ABB RobotStudio station: 210021601076.rspag

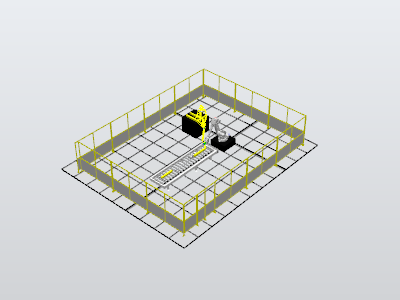
--- station ---
Station Aslam (saved by RobotStudio 23.2.10478.1)
Controller Controller2, task T_ROB1: task frame (RAPID world) sits at (580.05, 27.7, 395.4) mm, rotated rx 0 ry 0 rz 0.37 deg in the station
Controller Controller2
  mechanical unit ROB_1: IRB4600_40_255_C_01, 6 joints, base frame (0, 0, 0) mm
Layout (positions relative to the parent item):
  - Smart_Gripper_Servo_One_Vacuum [mechanism, from %ABB.RobotStudio.Models.SmartGripper%\ABB_Smart_Gripper_Servo_One_Vacuum.rslib] at (1934.43, -88.9, 888.73) mm, rotated rx -166.7 ry 89.28 rz -166.28 deg; joint values [0] (rad or m)
  - Conveyer [part, from %ABB.RobotStudio.Models.Conveyors%\Conveyor 950 4000 h2.rslib] at (1600, -500, 0) mm
  - Base [part] at (-3.62, 631.17, 0) mm, rotated rx 0 ry 0 rz 0.33 deg, size 1000 x 1000 x 400 mm
  - Box [part], size 800 x 100 x 100 mm
  - Conveyer [smart component]
      signals: DI movel, DO indic
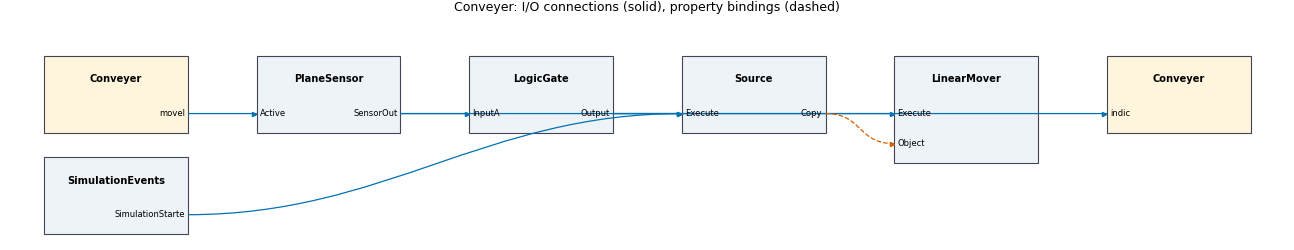
      connections:
        Conveyer.movel -> PlaneSensor.Active
        PlaneSensor.SensorOut -> Conveyer.indic
        PlaneSensor.SensorOut -> LogicGate.InputA
        LogicGate.Output -> LinearMover.Execute
        LogicGate.Output -> Source.Execute
        SimulationEvents.SimulationStarted -> Source.Execute
        Source.Copy => LinearMover.Object
    - PlaneSensor [smart component, from Components\PlaneSensor.rslib] at (1568.3, 52.45, 0) mm
        properties: Origin=[0.238634878927635 0.29755427370953 0.425]; Axis1=[0.1 0 0.1]; Axis2=[0 -0.77 0]; Tag=(none); SensedPart=Box_18
      - _sensorPart_ [part], size 100 x 770 x 100 mm
    - Source [smart component, from Components\Source.rslib]
        properties: Source=Box; Copy=Box_18; Parent=(none); Position=[0 0 0]; Orientation=[0 0 0]; Transient=false; PhysicsBehavior=-1
    - LinearMover [smart component, from Components\LinearMover.rslib]
        properties: Object=Box_18; Direction=[-3 0 0]; Speed=1; Reference=Global; ReferenceObject=(none)
    - LogicGate [smart component, from Components\LogicGate.rslib]
        properties: Operator=NOT; Delay=0
    - SimulationEvents [smart component, from Components\SimulationEvents.rslib]
  - AttachDetach [smart component]
      signals: DI attach, DO do
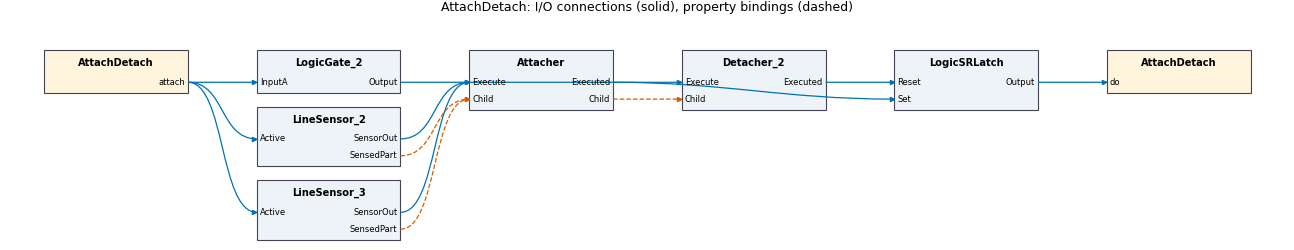
      connections:
        AttachDetach.attach -> LogicGate_2.InputA
        AttachDetach.attach -> LineSensor_2.Active
        LineSensor_2.SensorOut -> Attacher.Execute
        Detacher_2.Executed -> LogicSRLatch.Reset
        Attacher.Executed -> LogicSRLatch.Set
        LogicSRLatch.Output -> AttachDetach.do
        LogicGate_2.Output -> Detacher_2.Execute
        AttachDetach.attach -> LineSensor_3.Active
        LineSensor_3.SensorOut -> Attacher.Execute
        LineSensor_2.SensedPart => Attacher.Child
        Attacher.Child => Detacher_2.Child
        LineSensor_3.SensedPart => Attacher.Child
    - Attacher [smart component, from Components\Attacher.rslib]
        properties: Parent=Smart_Gripper_Servo_One_Vacuum; Flange=1; Child=Box_17; Mount=false; Offset=[0 0 0]; Orientation=[0 0 0]
    - Detacher_2 [smart component, from Components\Detacher.rslib]
        properties: Child=Box_17; KeepPosition=true
    - LogicSRLatch [smart component, from Components\LogicSRLatch.rslib]
    - LogicGate_2 [smart component, from Components\LogicGate.rslib]
        properties: Operator=NOT; Delay=0
    - LineSensor_3 [smart component, from Components\LineSensor.rslib] at (1971.18, -70.27, 838.23) mm, rotated rx -179.84 ry -0.7 rz -179.57 deg
        properties: Start=[0 0 0]; End=[0 0 0.02]; Length=0.02; Radius=0.0005; Tag=(none); SensedPart=Box_17; SensedPoint=[0.551275024414063 -1.6518037109375 1.09683813476563]
      - _sensorPart_ [part], size 1 x 1 x 20 mm
  - Box_ref2 [part] at (-4421.56, -1482.88, 580.2) mm, rotated rx 0 ry 0 rz -0.2 deg, size 800 x 100 x 100 mm
  - Place_box [part] at (0, -2580.03, 0) mm, size 1100 x 1100 x 1000 mm
  - Box_ref [part] at (986.59, 2917.03, 580.2) mm, rotated rx 0 ry 0 rz -90.6 deg, size 800 x 100 x 100 mm
  - IRB4600_40_255_C_01 [mechanism, from %ABB.RobotStudio.Models.IRB4600%\IRB4600_40_255_C_G_01.rslib] at (580.05, 27.7, 395.4) mm, rotated rx 0 ry 0 rz 0.37 deg; joint values [-0.1026, 0.2903, 0.8053, -3.2587, 1.0862, 3.1922] (rad or m)
  - Box_7 [part], size 800 x 100 x 100 mm
  - Box_9 [part], size 800 x 100 x 100 mm
  - Box_1 [part], size 800 x 100 x 100 mm
  - Box_3 [part], size 800 x 100 x 100 mm
  - Box_4 [part] at (638.69, 2911.14, 517.63) mm, rotated rx 0.12 ry -0.74 rz -90.21 deg, size 800 x 100 x 100 mm
  - Box_6 [part], size 800 x 100 x 100 mm
  - Box_7 [part], size 800 x 100 x 100 mm
  - Box_8 [part] at (-4416.13, -1490.91, 542.63) mm, rotated rx 0.37 ry -0.47 rz -0.11 deg, size 800 x 100 x 100 mm
  - Box_9 [part] at (953.48, 2910.35, 521.52) mm, rotated rx 0.12 ry -0.74 rz -90.21 deg, size 800 x 100 x 100 mm
  - Fence_2500 [graphiccomponentgroup, from Equipment\Fence_2500.rslib] at (-2465.89, 934.33, 0) mm
    - Body 1 [part, from Equipment\Fence_2500.rslib]
    - Body 2 [part, from Equipment\Fence_2500.rslib]
  - Fence_2500_2 [graphiccomponentgroup, from Equipment\Fence_2500.rslib] at (-2458.15, -1574.69, -2.82) mm
    - Body 1 [part, from Equipment\Fence_2500.rslib]
    - Body 2 [part, from Equipment\Fence_2500.rslib]
  - Fence_2500_3 [graphiccomponentgroup, from Equipment\Fence_2500.rslib] at (-2458.94, -4084.22, 0) mm
    - Body 1 [part, from Equipment\Fence_2500.rslib]
    - Body 2 [part, from Equipment\Fence_2500.rslib]
  - Fence_2500_4 [graphiccomponentgroup, from Equipment\Fence_2500.rslib] at (112.46, -4080.59, 0) mm, rotated rx 0 ry 0 rz -90 deg
    - Body 1 [part, from Equipment\Fence_2500.rslib]
    - Body 2 [part, from Equipment\Fence_2500.rslib]
  - Fence_2500_5 [graphiccomponentgroup, from Equipment\Fence_2500.rslib] at (2616.81, -4080.59, 0) mm, rotated rx 0 ry 0 rz -90 deg
    - Body 1 [part, from Equipment\Fence_2500.rslib]
    - Body 2 [part, from Equipment\Fence_2500.rslib]
  - Fence_2500_6 [graphiccomponentgroup, from Equipment\Fence_2500.rslib] at (-2390.88, -4080.59, 0) mm, rotated rx 0 ry 0 rz -90 deg
    - Body 1 [part, from Equipment\Fence_2500.rslib]
    - Body 2 [part, from Equipment\Fence_2500.rslib]
  - Fence_2500_7 [graphiccomponentgroup, from Equipment\Fence_2500.rslib] at (7575.33, -4087.76, 0) mm, rotated rx 0 ry 0 rz 90 deg
    - Body 1 [part, from Equipment\Fence_2500.rslib]
    - Body 2 [part, from Equipment\Fence_2500.rslib]
  - Fence_2500_8 [graphiccomponentgroup, from Equipment\Fence_2500.rslib] at (7396.23, 964.23, 0) mm
    - Body 1 [part, from Equipment\Fence_2500.rslib]
    - Body 2 [part, from Equipment\Fence_2500.rslib]
  - Fence_2500_9 [graphiccomponentgroup, from Equipment\Fence_2500.rslib] at (7396.23, -1514.89, 0) mm
    - Body 1 [part, from Equipment\Fence_2500.rslib]
    - Body 2 [part, from Equipment\Fence_2500.rslib]
  - Fence_2500_10 [graphiccomponentgroup, from Equipment\Fence_2500.rslib] at (7396.23, -4035.95, 0) mm
    - Body 1 [part, from Equipment\Fence_2500.rslib]
    - Body 2 [part, from Equipment\Fence_2500.rslib]
  - Gate [graphiccomponentgroup, from Equipment\Fence_Gate.rslib] at (5874.56, 3415.05, 0) mm, rotated rx 0 ry 0 rz -90 deg
    - Body 1 [part, from Equipment\Fence_Gate.rslib]
    - Body 2 [part, from Equipment\Fence_Gate.rslib]
    - Body 3 [part, from Equipment\Fence_Gate.rslib]
  - Fence_2500_11 [graphiccomponentgroup, from Equipment\Fence_2500.rslib] at (-2421.34, 3391.49, 0) mm, rotated rx 0 ry 0 rz -90 deg
    - Body 1 [part, from Equipment\Fence_2500.rslib]
    - Body 2 [part, from Equipment\Fence_2500.rslib]
  - Fence_2500_12 [graphiccomponentgroup, from Equipment\Fence_2500.rslib] at (112.89, 3391.49, 0) mm, rotated rx 0 ry 0 rz -90 deg
    - Body 1 [part, from Equipment\Fence_2500.rslib]
    - Body 2 [part, from Equipment\Fence_2500.rslib]
  - Fence_2500_13 [graphiccomponentgroup, from Equipment\Fence_2500.rslib] at (2639.04, 3391.49, 0) mm, rotated rx 0 ry 0 rz -90 deg
    - Body 1 [part, from Equipment\Fence_2500.rslib]
    - Body 2 [part, from Equipment\Fence_2500.rslib]
  - Fence_740_2 [graphiccomponentgroup, from Equipment\Fence_740.rslib] at (5139.35, 3403.98, 0) mm, rotated rx 0 ry 0 rz -90 deg
    - Body 1 [part, from Equipment\Fence_740.rslib]
    - Body 2 [part, from Equipment\Fence_740.rslib]
  - Box_13 [part], size 800 x 100 x 100 mm
  - Box_14 [part] at (-2520, 0, 0) mm, size 800 x 100 x 100 mm
  - Box_15 [part] at (-4416.13, -1490.91, 542.63) mm, rotated rx 0.37 ry -0.47 rz -0.11 deg, size 800 x 100 x 100 mm
  - Box_16 [part] at (953.48, 2910.35, 521.52) mm, rotated rx 0.12 ry -0.74 rz -90.21 deg, size 800 x 100 x 100 mm
  - Box_17 [part] at (638.69, 2911.14, 517.63) mm, rotated rx 0.12 ry -0.74 rz -90.21 deg, size 800 x 100 x 100 mm
  - Box_18 [part] at (-2664, 0, 0) mm, size 800 x 100 x 100 mm
Attachment: LineSensor_3 is attached to Smart_Gripper_Servo_One_Vacuum / DownFinger
Attachment: Smart_Gripper_Servo_One_Vacuum is attached to IRB4600_40_255_C_01 / Link6
Station logic (signal -> signal, property => property):
  Controller2.out -> AttachDetach.attach
  Controller2.di_output -> Conveyer.movel
  Conveyer.indic -> Controller2.start

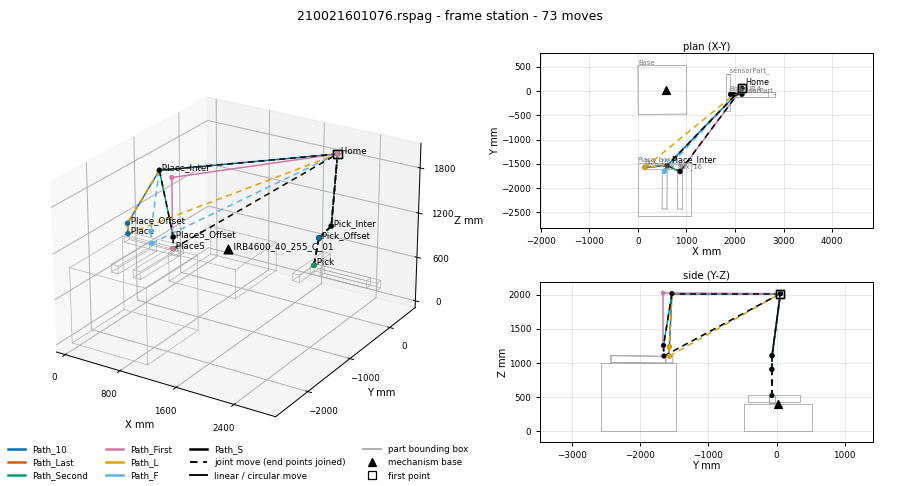
[picture p0: tool path of 210021601076.rspag in frame station, 73 of 73 moves have a stored position in this frame; points joined in program order, loops and branches not executed]
--- Controller Data/Controller2/RAPID/TASK1/PROGMOD/CalibData.mod ---
MODULE CalibData
    PERS tooldata Servo:=[TRUE,[[0,0,84],[1,0,0,0]],[0.226,[8.9,12.3,48.7],[1,0,0,0],0.00021,0.00024,0.00009]];
    PERS tooldata VaccumOne:=[TRUE,[[63.5,18.5,37.5],[0.707106781,0,0.707106781,0]],[0.226,[8.9,12.3,48.7],[1,0,0,0],0.00021,0.00024,0.00009]];
ENDMODULE

--- Controller Data/Controller2/RAPID/TASK1/PROGMOD/Module1.mod ---
MODULE Module1
        CONST robtarget Home:=[[1562.639382153,18.5,1623.75738686],[0.258819046,0,-0.965925826,0],[-1,-1,0,1],[9E+09,9E+09,9E+09,9E+09,9E+09,9E+09]];
    CONST robtarget Pick:=[[1325.709206308,-105.69931637,127.507161245],[0.005604326,-0.000424517,-0.99998295,0.001584379],[-1,-3,2,0],[9E+09,9E+09,9E+09,9E+09,9E+09,9E+09]];
    CONST robtarget Pick_Inter:=[[1561.851467861,-103.162107412,713.081838562],[0.258819024,0,-0.965925832,0],[-1,-3,2,0],[9E+09,9E+09,9E+09,9E+09,9E+09,9E+09]];
    CONST robtarget Pick_Offset:=[[1391.779201858,-106.126964158,512.226578953],[0.005604378,-0.000424533,-0.99998295,0.001584379],[-1,-3,2,0],[9E+09,9E+09,9E+09,9E+09,9E+09,9E+09]];
    CONST robtarget Place_Inter:=[[11.867363508,-1562.703465576,1623.756983637],[0.182623873,-0.68446068,-0.681561662,-0.183400653],[-2,-3,2,1],[9E+09,9E+09,9E+09,9E+09,9E+09,9E+09]];
    CONST robtarget Place:=[[-440.70574459,-1597.548111643,707.1200986],[0.001483954,-0.00137647,-0.999996574,-0.001659987],[-2,-2,0,1],[9E+09,9E+09,9E+09,9E+09,9E+09,9E+09]];
    CONST robtarget Place_Offset:=[[-444.124698969,-1597.525985837,843.908044243],[0.001483948,-0.001376451,-0.999996574,-0.001659976],[-2,-2,0,1],[9E+09,9E+09,9E+09,9E+09,9E+09,9E+09]];
    CONST robtarget PlaceS_Offset:=[[280.069318323,-1687.384959127,863.62826548],[0.000238405,0.708711216,0.705497899,-0.001034476],[-1,-2,1,0],[9E+09,9E+09,9E+09,9E+09,9E+09,9E+09]];
    CONST robtarget PlaceS:=[[275.144596365,-1682.104959802,708.235040947],[0.000238464,0.708711109,0.705498006,-0.001034365],[-1,-2,1,0],[9E+09,9E+09,9E+09,9E+09,9E+09,9E+09]];
    CONST robtarget PlaceF_Inter:=[[275.646442284,-1694.12601053,1633.167957717],[0.000238738,0.70871119,0.705497925,-0.00103415],[-1,-4,3,1],[9E+09,9E+09,9E+09,9E+09,9E+09,9E+09]];
    CONST robtarget PlaceF_Offset:=[[275.646447462,-1694.126005121,854.024783097],[0.000238763,0.708711188,0.705497927,-0.001034117],[-1,-4,3,1],[9E+09,9E+09,9E+09,9E+09,9E+09,9E+09]];
    CONST robtarget Place_F:=[[275.686493171,-1687.929599777,709.019601147],[0.000238779,0.708711216,0.705497899,-0.001034127],[-1,-4,3,1],[9E+09,9E+09,9E+09,9E+09,9E+09,9E+09]];
    CONST robtarget Place2_Offset:=[[-43.343867547,-1685.291053434,863.62834295],[0.000238739,0.708711198,0.705497917,-0.001034153],[-2,-3,2,0],[9E+09,9E+09,9E+09,9E+09,9E+09,9E+09]];
    CONST robtarget Place2:=[[-39.637509275,-1679.274249515,704.345546214],[0.000238825,0.708711224,0.705497891,-0.001034082],[-2,-3,2,0],[9E+09,9E+09,9E+09,9E+09,9E+09,9E+09]];
!***********************************************************
    !
    ! Module:  Module1
    !
    ! Description:
    !   <Insert description here>
    !
    ! Author: shahu
    !
    ! Version: 1.0
    !
    !***********************************************************


    !***********************************************************
    !
    ! Procedure main
    !
    !   This is the entry point of your program
    !
    !***********************************************************
    PROC main()
        !Add your code here
    ENDPROC
    PROC Path_10()
        MoveJ Home,v1000,z100,VaccumOne\WObj:=wobj0;
        MoveJ Pick_Inter,v1000,z100,VaccumOne\WObj:=wobj0;
        MoveJ Pick_Offset,v1000,z100,VaccumOne\WObj:=wobj0;
        MoveJ Pick,v1000,z100,VaccumOne\WObj:=wobj0;
        MoveJ Pick_Offset,v1000,z100,VaccumOne\WObj:=wobj0;
        MoveJ Pick_Inter,v1000,z100,VaccumOne\WObj:=wobj0;
        MoveJ Home,v1000,z100,VaccumOne\WObj:=wobj0;
        MoveL Place_Inter,v1000,z100,VaccumOne\WObj:=wobj0;
        MoveL Place_Offset,v1000,z100,VaccumOne\WObj:=wobj0;
        MoveL Place,v1000,z100,VaccumOne\WObj:=wobj0;
    ENDPROC
    PROC Path_Last()
        MoveJ Home,v1000,z100,VaccumOne\WObj:=wobj0;
        MoveJ Pick_Inter,v1000,z100,VaccumOne\WObj:=wobj0;
        MoveJ Pick_Offset,v1000,z100,VaccumOne\WObj:=wobj0;
        MoveJ Pick,v1000,z100,VaccumOne\WObj:=wobj0;
        MoveJ Pick_Offset,v1000,z100,VaccumOne\WObj:=wobj0;
        MoveJ Pick_Inter,v1000,z100,VaccumOne\WObj:=wobj0;
        MoveJ Home,v1000,z100,VaccumOne\WObj:=wobj0;
        MoveJ Place_Inter,v1000,z100,VaccumOne\WObj:=wobj0;
        MoveJ Place_Offset,v1000,z100,VaccumOne\WObj:=wobj0;
        MoveJ Place,v1000,z100,VaccumOne\WObj:=wobj0;
    ENDPROC
    PROC Path_Second()
        MoveJ Home,v1000,z100,VaccumOne\WObj:=wobj0;
        MoveJ Pick_Inter,v1000,z100,VaccumOne\WObj:=wobj0;
        MoveJ Pick_Offset,v1000,z100,VaccumOne\WObj:=wobj0;
        MoveJ Pick,v1000,z100,VaccumOne\WObj:=wobj0;
        MoveJ Pick_Offset,v1000,z100,VaccumOne\WObj:=wobj0;
        MoveJ Pick_Inter,v1000,z100,VaccumOne\WObj:=wobj0;
        MoveJ Home,v1000,z100,VaccumOne\WObj:=wobj0;
        MoveJ Place_Inter,v1000,z100,VaccumOne\WObj:=wobj0;
        MoveL PlaceS_Offset,v1000,z100,VaccumOne\WObj:=wobj0;
        MoveJ PlaceS,v1000,z100,VaccumOne\WObj:=wobj0;
    ENDPROC
    PROC Path_First()
        MoveJ Home,v1000,z100,VaccumOne\WObj:=wobj0;
        MoveJ Pick_Inter,v1000,z100,VaccumOne\WObj:=wobj0;
        MoveJ Pick_Offset,v1000,z100,VaccumOne\WObj:=wobj0;
        MoveJ Pick,v1000,z100,VaccumOne\WObj:=wobj0;
        MoveJ Pick_Offset,v1000,z100,VaccumOne\WObj:=wobj0;
        MoveJ Pick_Inter,v1000,z100,VaccumOne\WObj:=wobj0;
        MoveJ Home,v1000,z100,VaccumOne\WObj:=wobj0;
        MoveL PlaceF_Inter,v1000,z100,VaccumOne\WObj:=wobj0;
        MoveL PlaceF_Offset,v1000,z100,VaccumOne\WObj:=wobj0;
        MoveJ Place_F,v1000,z100,VaccumOne\WObj:=wobj0;
    ENDPROC
    PROC Final_Path()
        Path_F;
        Path_L;
        Path_S;

    ENDPROC
    PROC Path_L()
        MoveJ Home,v1000,z100,VaccumOne\WObj:=wobj0;
        MoveJ Pick_Inter,v1000,z100,VaccumOne\WObj:=wobj0;
        MoveJ Pick_Offset,v1000,z100,VaccumOne\WObj:=wobj0;
        MoveJ Pick,v1000,z100,VaccumOne\WObj:=wobj0;
        WaitTime 1;
        SetDO out,1;
        WaitTime 1;
        MoveJ Pick_Offset,v1000,z100,VaccumOne\WObj:=wobj0;
        MoveJ Pick_Inter,v1000,z100,VaccumOne\WObj:=wobj0;
        MoveJ Home,v1000,z100,VaccumOne\WObj:=wobj0;
        MoveJ Place_Inter,v1000,z100,VaccumOne\WObj:=wobj0;
        MoveJ Place_Offset,v1000,z100,VaccumOne\WObj:=wobj0;
        MoveJ Place,v1000,z100,VaccumOne\WObj:=wobj0;
        WaitTime 1;
        SetDO out,0;
        WaitTime 1;
        MoveJ Home,v1000,z100,VaccumOne\WObj:=wobj0;
    ENDPROC
    PROC Path_F()
        MoveJ Home,v1000,z100,VaccumOne\WObj:=wobj0;
        MoveJ Pick_Inter,v1000,z100,VaccumOne\WObj:=wobj0;
        MoveJ Pick_Offset,v1000,z100,VaccumOne\WObj:=wobj0;
        MoveJ Pick,v1000,z100,VaccumOne\WObj:=wobj0;
        WaitTime 1;
        SetDO out,1;
        WaitTime 1;
        MoveJ Pick_Offset,v1000,z100,VaccumOne\WObj:=wobj0;
        MoveJ Pick_Inter,v1000,z100,VaccumOne\WObj:=wobj0;
        MoveJ Home,v1000,z100,VaccumOne\WObj:=wobj0;
        MoveJ Place_Inter,v1000,z100,VaccumOne\WObj:=wobj0;
        MoveJ Place2_Offset,v1000,z100,VaccumOne\WObj:=wobj0;
        MoveJ Place2,v1000,z100,VaccumOne\WObj:=wobj0;
        WaitTime 1;
        SetDO out,0;
        WaitTime 1;
        MoveJ Home,v1000,z100,VaccumOne\WObj:=wobj0;
    ENDPROC
    PROC Path_S()
        MoveJ Home,v1000,z100,VaccumOne\WObj:=wobj0;
        MoveJ Pick_Inter,v1000,z100,VaccumOne\WObj:=wobj0;
        MoveJ Pick_Offset,v1000,z100,VaccumOne\WObj:=wobj0;
        MoveJ Pick,v1000,z100,VaccumOne\WObj:=wobj0;
        WaitTime 1;
        SetDO out,1;
        WaitTime 1;
        MoveJ Pick_Offset,v1000,z100,VaccumOne\WObj:=wobj0;
        MoveJ Pick_Inter,v1000,z100,VaccumOne\WObj:=wobj0;
        MoveJ Home,v1000,z100,VaccumOne\WObj:=wobj0;
        MoveJ Place_Inter,v1000,z100,VaccumOne\WObj:=wobj0;
        MoveJ PlaceS_Offset,v1000,z100,VaccumOne\WObj:=wobj0;
        MoveJ PlaceS,v1000,z100,VaccumOne\WObj:=wobj0;
        WaitTime 1;
        SetDO out,0;
        WaitTime 1;
        MoveJ Home,v1000,z100,VaccumOne\WObj:=wobj0;
    ENDPROC
ENDMODULE

--- Controller Data/Controller2/SYSPAR/EIO.cfg ---
EIO:CFG_1.0:6:1::
#
EIO_SIGNAL:

      -Name "out" -SignalType "DO"

      -Name "di_output" -SignalType "DO"

      -Name "start" -SignalType "DI"
